Universal Robots PolyScope program: AlvarezZavaleta-LuisAlberto-P2.urp

Program AlvarezZavaleta-LuisAlberto-P2 (installation=default directory=/home/ur/ursim-current/programs/sf_vagrant createdIn=5.14.5 lastSavedIn=5.14.5 robotSerialNumber=20195399999)
Calibrated DH parameters: a=[0, -0.24355, -0.2132, 0, 0, 0]; d=[0.15185, 0, 0, 0.13105, 0.08535, 0.0921]; alpha=[1.570796, 0, 0, 1.570796, -1.570796, 0]; deltaTheta=[0, 0, 0, 0, 0, 0]
InitVariablesNode
Robot Program (runOnlyOnce=true)
  y := -50
  rx := 0
  ry := 0
  rz := 0
  P_ini := get_actual_tcp_pose()
  desplazamiento := p[0,y/1000,0,rx,ry,rz]
  pos_coger := pose_add(P_ini, desplazamiento)
  z := -100
  desplazamiento := p[0,0,z/1000,0,0,0]
  PrimerPunto := pose_add(pos_coger, desplazamiento)
  y := -140
  desplazamiento := p[0,y/1000,0,0,0,0]
  SegundoPunto := pose_add(PrimerPunto, desplazamiento)
  x := -130
  desplazamiento := p[x/1000,0,0,0,0,0]
  TercerPunto := pose_add(PrimerPunto, desplazamiento)
  y := -30
  desplazamiento := p[0,y/1000,0,0,0,0]
  CuartoPunto := pose_add(SegundoPunto, desplazamiento)
  x := -50
  desplazamiento := p[x/1000,0,0,0,0,0]
  QuintoPunto := pose_add(TercerPunto, desplazamiento)
  MoveJ speed 60 deg/s, acceleration 80 deg/s^2 (useActiveTCP=true) feature=Base
    Wait Sleep waitTime=1
    Waypoint Variable (Variable): motionParameters(blendRadius=0.05); variable=pos_coger
    Waypoint Variable (Variable): variable=PrimerPunto
    Loop Counting (count=2) loopVariable(name=Loop_1)
      MoveL speed 250 mm/s, acceleration 1200 mm/s^2 (useActiveTCP=true) feature=Base
        Waypoint Variable (Variable): variable=SegundoPunto
        Waypoint Variable (Variable): variable=TercerPunto
        Waypoint Variable (Variable): variable=PrimerPunto
    Loop Counting (count=2) loopVariable(name=Loop_2)
      Waypoint Variable (Variable): variable=CuartoPunto
      Waypoint Variable (Variable): variable=QuintoPunto
      Waypoint Variable (Variable): variable=PrimerPunto
